// TIA Portal V17 export
// export: Created 2025-03-13T10:30:37.6323165Z, ExportSetting WithDefaults, DisplayName Totally Integrated Automation Portal, DisplayVersion V17 Update 8, DisplayName TIA Portal Openness, DisplayVersion V17 Update 8, DisplayName TIA Portal Version Control Interface, DisplayVersion V17, DisplayName SINAMICS Startdrive Advanced, DisplayVersion V17 SP2, DisplayName SINAMICS Startdrive G110M, G120, G120C, G120D, G120P, G115D, DisplayVersion V17 SP2, DisplayName SINAMICS Startdrive G130, G150, S120, S150, SINAMICS MV, S210, DisplayVersion V17 SP2, DisplayName STEP 7 Professional, DisplayVersion V17 Update 8, DisplayName SINUMERIK ONE STEP 7 Toolbox, DisplayVersion V17 Update 12, DisplayName SINUMERIK 840D sl STEP 7 Toolbox, DisplayVersion V17 Update 12, DisplayName STEP 7 Safety, DisplayVersion V17 Update 6, DisplayName WinCC Advanced, DisplayVersion V17 Update 8
DATA_BLOCK "DB8100_MANUAL_LOADING_PART_STATUS"   // DB8100
{ S7_Optimized_Access := 'FALSE'; DB_Accessible_From_OPC_UA := 'FALSE' }
VERSION : 0.1
// stored: AutoNumber false, DBAccessibleFromOPCUA false, DBAccessibleFromWebserver true, IsOnlyStoredInLoadMemory false, IsWriteProtectedInAS false
   VAR
      UNIT_01_DELETE_PART_HMI_BUTTON : Bool;   // DELETE PART FROM FIXTURE IN UNIT 01 STATION 1 HMI BUTTON
      UNIT_01_ADD_PART_HMI_BUTTON : Bool;   // ADD PART TO FIXTURE IN UNIT 01 STATION 1 HMI BUTTON
      UNIT_01_SKIP_LOADING_FIX_STA_1_HMI_BUTTON : Bool;   // UNIT 01 SKIP LOADING FIXTURE IN STATION 1 HMI BUTTON
      UNIT_01_NO_FACE_R_PARTS_TO_DELIVER : Bool;   // NO FACE R PARTS TO DELIVER UNIT 01
      UNIT_01_NO_FACE_N_PARTS_TO_DELIVER : Bool;   // NO FACE N PARTS TO DELIVER UNIT 01
      UNIT_01_SPARE_3 : Bool;
      UNIT_01_SPARE_4 : Bool;
      UNIT_01_SPARE_5 : Bool;
      UNIT_02_DELETE_PART_HMI_BUTTON : Bool;   // DELETE PART FROM FIXTURE IN UNIT 02 STATION 1 HMI BUTTON
      UNIT_02_ADD_PART_HMI_BUTTON : Bool;   // ADD PART TO FIXTURE IN UNIT 02 STATION 1 HMI BUTTON
      UNIT_02_SKIP_LOADING_FIX_STA_1_HMI_BUTTON : Bool;   // UNIT 02 SKIP LOADING FIXTURE IN STATION 1 HMI BUTTON
      UNIT_02_NO_FACE_R_PARTS_TO_DELIVER : Bool;   // NO FACE R PARTS TO DELIVER UNIT 02
      UNIT_02_NO_FACE_N_PARTS_TO_DELIVER : Bool;   // NO FACE N PARTS TO DELIVER UNIT 02
      UNIT_02_SPARE_3 : Bool;
      UNIT_02_SPARE_4 : Bool;
      UNIT_02_SPARE_5 : Bool;
      UNIT_03_DELETE_PART_HMI_BUTTON : Bool;   // DELETE PART FROM FIXTURE IN UNIT 03 STATION 1 HMI BUTTON
      UNIT_03_ADD_PART_HMI_BUTTON : Bool;   // ADD PART TO FIXTURE IN UNIT 03 STATION 1 HMI BUTTON
      UNIT_03_SPARE_1 : Bool;
      UNIT_03_SPARE_2 : Bool;
      UNIT_03_SPARE_3 : Bool;
      UNIT_03_SPARE_4 : Bool;
      UNIT_03_SPARE_5 : Bool;
      UNIT_03_SPARE_6 : Bool;
   END_VAR
BEGIN
END_DATA_BLOCK
